// TIA Portal V18 export
FUNCTION "pump RPM" : Void   // FC28, LAD
{ S7_Optimized_Access := 'TRUE' }
VERSION : 0.1
// stored: AutoNumber true, IsIECCheckEnabled false, SetENOAutomatically false, UDAEnableTagReadback false
BEGIN

REGION Network 1 (SCL)
   "RPM".A := ((DINT_TO_REAL("RPM PUMP A")) / "Pump & Flowrate"."Pump A"."speed sensor impulse") * 60.0;
   "RPM".B := ((DINT_TO_REAL("RPM PUMP B")) / "Pump & Flowrate"."Pump B"."speed sensor impulse") * 60.0;

   "RPM"."a selected" := ("RPM"."speed sensor selection A" = 1);
   "RPM"."b selected" := ("RPM"."speed sensor selection B" = 1);
   "RPM"."ab selected" := "RPM"."a selected" OR "RPM"."b selected";
END_REGION
END_FUNCTION
